// TIA Portal V20 export
TYPE "RollerConvConfig"
   STRUCT
      DeadEnd : Bool;   // Dead End Disable Positiong Fault
      TrspNoLowSpeed : Bool;   // Input 14
      StopDetSetUsed : Bool;   // Input 0
      LowSpeedDetSetUsed : Bool;   // Low Speed Det Used
      LowSpeedDetSetConstOn : Bool;   // Low Speed Sensor Constant on
      StopDetResUsed : Bool;   // Stop detection Reset used
      LowSpeedDetResUsed : Bool;   // Input 10
      LowSpeedDetResConstOn : Bool;   // Lowspeed stop detection Constant On
      TrainActivatedSet : Bool;   // Train transport used set direction
      TrfInSetUsed : Bool;   // Transfer In Set Used
      TrfOutSetUsed : Bool;   // Transfer Out Reset Used
      TrainActivatedRes : Bool;   // Train transport used Reset direction
      TrfInResUsed : Bool;   // Transfer In Reset Used
      TrfOutResUsed : Bool;   // Transfer Out Reset Used
      EnableAlarmHW : Bool := TRUE;   // Enable Alarm hardware (e.g. Safetyswitch, Motorprotector, detections)
      EnableAlarmTransfer : Bool;   // Enable Alarm transfer (e.g. Transfer in , transfer out)
      EnableG120Reset : Bool;   // Enable Driver Reset
      EnableCheckSpeedOK : Bool;   // Enable Speed checking on the G120 Driver
      EnableSetpoint : Bool;   // Enable setpoint
      EnableRFG : Bool;   // Follow setpoint
      NotQuickStop : Bool;   // QuickStop function; When FALSE the QuickStop of the G120 is Active
      NotImmediateStop : Bool;   // Immediate function; When FALSE the immediate stop of the G120 is Active
      EnableBeltControlSetDet : Bool;   // Config Belt Control
      EnableBeltControlResDet : Bool;   // Config Belt Control
      SLSUsed : Bool;   // Profisafe SLS Configuration Used
      SafetySwUsed : Bool;   // Input 12
      SafetySwNc : Bool;   // Input 15
      ReleaseBrakeUsed : Bool;   // Input 13
      RearDetUsed : Bool;   // Input 9
      RevSwUsed : Bool;   // Input 8
      MotorProtectionUsed : Bool;   // Motorprotection Used
      MotorProtectionNc : Bool;   // Motorprotection NC
      InitDirection : Bool;   // Input 6
      ForceManual : Bool;   // Configuration
      Spare1 : Bool;   // Spare
      Spare2 : Bool;   // Spare
      Spare3 : Bool;   // Spare
      TrfMaxTime : DInt;   // Max allowed transfertime (millisec)
      RPMSpeed : Real;   // Movment Rpm
      EnableRPMSpeed : Bool;   // Enable RPM Speed
      ReferenceSpeed : Int;   // Reference value for speed, stored in P2000 ot the SINAMICS
      ReferenceCurrent : Real;   // Reference value for current, stored in P2002 ot the SINAMICS
      ReferenceTorque : Real;   // Reference value for torque, stored in P2003 ot the SINAMICS
      DelaySetStopDet : Time := T#1ms;   // Delay Time Stop Detection
      DelayResStopDet : Time := T#1ms;   // Delay Time Stop Detection
      HWSubInput : HW_SUBMODULE;   // Address (input/output)
      HWSubOutput : HW_SUBMODULE;   // I/O
      SafetyAddress : HW_SUBMODULE;   // Address (input/output)
      FilterBeltControlSec : DInt;   // Filter In Seconds Belt Control
   END_STRUCT;
END_TYPE
